INTERFACE ITF_ObslugaAlarmow_Podzespol EXTENDS ITF_ObslugaAlarmow_ElementWykonawczy

END_INTERFACE

(* stored: Version 1.1.0.1, ProductVersion 3.1.4024.11
   Itf ITF_ObslugaAlarmow_Podzespol: Id {bcbecd20-91cf-4531-aaec-a94558b8febc} *)
